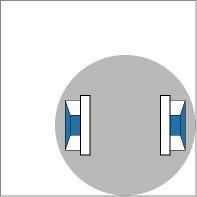
VISUALIZATION VISU_Tube_Top_fork  // 197x197
VAR_IN_OUT
	azi : LREAL;
END_VAR
    Ellipse (55,55 140x140)
    Rectangle (160,95 10x60)
        p2858320360: azi
    Rectangle (80,95 10x60)
        p2858320360: azi
    Polygon (170,100) (185,100) (180,115) (170,115)
        p2858320360: azi
    Polygon (170,150) (185,150) (180,135) (170,135)
        p2858320360: azi
    Polygon (180,135) (185,150) (185,100) (180,115)
        p2858320360: azi
    Polygon (170,135) (180,135) (180,115) (170,115)
        p2858320360: azi
    Polygon (65,100) (80,100) (80,115) (70,115)
        p2858320360: azi
    Polygon (65,150) (80,150) (80,130) (70,130)
        p2858320360: azi
    Polygon (65,100) (65,150) (70,135) (70,115)
        p2858320360: azi
    Polygon (70,135) (80,135) (80,115) (70,115)
        p2858320360: azi
END_VISUALIZATION

(* stored: Version 1.1.0.1, ProductVersion 3.1.4018.5
   Visu VISU_Tube_Top_fork: Id {c5f3ac08-86db-456d-b81a-1d6030b4b923} *)
